INTERFACE I_LinkSettings

PROPERTY PUBLIC DestinationId : NodeId
GET
END_GET
END_PROPERTY

PROPERTY PUBLIC DestinationPortId : PortId
GET
END_GET
END_PROPERTY

PROPERTY PUBLIC Id : T_MAXSTRING
GET
END_GET
END_PROPERTY

PROPERTY SourceId : NodeId
GET
END_GET
END_PROPERTY

PROPERTY PUBLIC SourcePortId : PortId
GET
END_GET
END_PROPERTY

END_INTERFACE

(* stored: Version 1.1.0.1, ProductVersion 3.1.4024.12
   Itf I_LinkSettings: Id {08907437-7ef4-003d-3793-9239ea2b7c04}
   Property DestinationId: Id {3937ae85-5bb6-0884-3ce8-f1549db5687e}
   Get Get: Id {c2d9ba1c-30ba-0746-22c0-4a1611e6eb99}
   Property DestinationPortId: Id {06043390-ce54-0b3b-3673-0637911b9648}
   Get Get: Id {7eb5ca01-eb3e-0f8f-36b6-3d7fab74d57a}
   Property Id: Id {652dd274-2840-098e-2266-c453e39cbfdf}
   Get Get: Id {f633d26c-9260-06e3-34ad-2c867522c6ef}
   Property SourceId: Id {11226632-74f3-06b9-179c-749e74957fbe}
   Get Get: Id {d985f42b-da47-08bd-3365-d0b0c3bd6a67}
   Property SourcePortId: Id {50699104-2f07-0615-0eeb-4187ac02e054}
   Get Get: Id {d65033b3-0873-0357-28ce-e5cc87b4252c} *)
